(* PLC project analog_pump, Dassault Systèmes ControlBuild 2024x *)
(* stored: creationDateTime 2023-10-03T11:13:00-01:00 *)

(* This module simulates the behaviour of an analog pump and its electrical control logic. *)
FUNCTION_BLOCK equipment_library.analog_pump
  VAR_INPUT
    voltage380 : BOOL := true;
    cmdSupply : BOOL := true;
    sensorSupply : BOOL := true;
  END_VAR
  VAR_INPUT
    onCmd : BOOL := false;
    setpoint : REAL := 0.0;
  END_VAR
  VAR_INPUT
    inputFlow : REAL := 0.0;
  END_VAR
  VAR_OUTPUT
    onFB : BOOL := false;
    thermal : BOOL := false;
  END_VAR
  VAR_OUTPUT
    speedVal : REAL := 0.0;
    outputFlow : REAL := 0.0;
  END_VAR
  VAR
    increment : REAL := 0.0;
    onState : BOOL := false;
    unit : REAL := 0.0;
    speedSetpoint : REAL := 0.0;
  END_VAR
  VAR CONSTANT
    nominalTime : REAL := 2.0;
    thermalLogic : BOOL := false;
    onFbLogic : BOOL := true;
    nominalSpeed : REAL := 3600.0;
    flowMax : REAL := 10000.0;
    flowPerHour : BOOL := true;
    flowPerMinute : BOOL := false;
  END_VAR
  VAR
    d_locking : BOOL := false;
    v_d_locking : REAL := 0.0;
    d_flow : BOOL := false;
    v_d_flow : REAL := 0.0;
    d_electrical : BOOL := false;
    v_d_electrical : BOOL := false;
    d_onFB : BOOL := false;
    v_d_onFB : BOOL := false;
  END_VAR


ACTION C_source_code:
/* -----------------------------------------------------------------	*/
/* Type : Model of Operative Behaviour					*/
/* Catégorie :   batch							*/
/* Author : Dassault Systemes						*/
/* Update date : June 2018							*/
/* -----------------------------------------------------------------	*/
/* This module simulates the behaviour of an analog pump and its 	*/
/* electrical control logic.						*/
/* ----------------------------------------------------------------	*/


/* ----------------------------------------------------------------	*/
/* Management of orders from Control Part					*/
/*	if there is no power supply for command 				*/
/*     the contactor doesn't understand the control order		*/
/* The setpoint can go from 0% up to +100%
/* ----------------------------------------------------------------	*/
if (d_electrical) 
	onState=v_d_electrical;
else
	onState = onCmd & cmdSupply & voltage380;

/* ----------------------------------------------------------------	*/
/* Management of  the rotation speed					*/
/* ----------------------------------------------------------------	*/
if (d_locking)  speedVal = v_d_locking;
else {
	/* Compute the increment of speed according to the simulation clock	*/
	if (nominalTime > 0.0)
		increment = (nominalSpeed / nominalTime) * (CLOCK_PERIOD/1000000.0);

	/* Compute the rotation speed setpoint	*/
	if (onState && (setpoint >=0.0) &&  (setpoint <= 100.0)) speedSetpoint = (setpoint / 100.0) * nominalSpeed;
	if (! onState) speedSetpoint = 0.0;
	
	/* Compute the speed ramp	*/
	if ( speedVal < speedSetpoint ) {
		speedVal += increment;
		if (speedVal > speedSetpoint)  speedVal = speedSetpoint;
	}
	if ( speedVal > speedSetpoint ) {
		speedVal -= increment;
		if (speedVal < speedSetpoint)  speedVal = speedSetpoint;
	}
}

/* ----------------------------------------------------------------	*/
/* Management of the thermal feedback					*/
/* ----------------------------------------------------------------	*/
if (d_electrical) thermal = v_d_electrical;
else
	thermal = ! thermalLogic && sensorSupply;

/* ----------------------------------------------------------------	*/
/* Management of feedback to Control Part					*/
/*     if a fault is required, the contactor feed-back 		*/
/*		 takes a preset state.					*/
/*	if there is no power supply for sensors 				*/
/*         contactor feed-back returns nothing				*/
/*     else contactor feed-back returns the contactor state combined	*/
/*	    with wiring logic.						*/
/* ----------------------------------------------------------------	*/
if (d_onFB) onFB = v_d_onFB;
else
	onFB = (onCmd ^ ! onFbLogic) && sensorSupply;

/* ----------------------------------------------------------------	*/
/* Management of the flow at the outlet of the pump			*/
/* The flow is computed according to the rotation speed of the pump	*/
/* and the flow at the inlet of the pump.					*/
/* This theorical flow rate is upper bounded with the maximal 	*/
/* manufacturer's flow.							*/
/* ----------------------------------------------------------------	*/
if (d_flow)
	outputFlow = v_d_flow;
else {
	if (nominalSpeed  > 0.0) {	
		if (flowPerHour) unit = 3600.0;
		else if (flowPerMinute) unit = 60.0;
			else unit = 1.0;
			
		outputFlow = ((flowMax * CLOCK_PERIOD / 1000000)  / unit) * (speedSetpoint / nominalSpeed  );
		if (outputFlow > inputFlow) outputFlow = inputFlow;		
	}
	else outputFlow =0.0;
}
END_ACTION
END_FUNCTION_BLOCK
